GLOBALCONSTANTS myOpcUaAddresses (* Global constants *)
  (* Standard: 61499-1; Description: Copyright (c) 2026 Meisterschulen am Ostbahnhof This program and the accompanying materials are made available under the terms of the Eclipse Public License 2.0 which is available at https://www.eclipse.org/legal/epl-2.0/ SPDX-License-Identifier: EPL-2.0 *)
  (* Version 1.0, 2026-09-02, Franz Höpfinger, Meisterschulen am Ostbahnhof *)
  PACKAGE VV::const::OPC_UA;
  VAR_GLOBAL CONSTANT
    Q1_LOCAL_READ : WSTRING := "opc_ua[READ;/Objects/DigitalOutput/Q1,1:s=Output_Q1]"; (* Geraet B (Station 12): lokal ueberwachter Knoten fuer Output_Q1 (ACTION=READ, passend zu AX_SUBSCRIBE_1 - siehe 4diac-Doku opcua.adoc Tabelle: Local/READ/SUBSCRIBE), von Geraet A per CLIENT_1_0 remote beschrieben *)
    Q1_REMOTE_WRITE : WSTRING := "opc_ua[WRITE;opc.tcp://192.168.1.12:4840#;/Objects/DigitalOutput/Q1,1:s=Output_Q1]"; (* Geraet A (Station 11): aktiver Remote-Write ueber CLIENT_1_0 auf denselben Knoten wie Q1_LOCAL_READ auf Geraet B (ACTION=WRITE, passend zu CLIENT - Remote/WRITE/CLIENT) - Pfad/Name-Suffix muss identisch bleiben, IP muss als Literal dupliziert werden (kein Verweis auf Computers.gcf moeglich) *)
    FF1_TRIGGER_LOCAL_READ : WSTRING := "opc_ua[READ;/Objects/ToggleFF/FF1_Trigger,1:s=FF1_Trigger]"; (* Geraet B (Station 12): lokal ueberwachter Trigger-Knoten (ACTION=READ, passend zu AX_SUBSCRIBE_1 - Local/READ/SUBSCRIBE), von Geraet A per CLIENT_1_0 remote beschrieben, um SoftKey_F1-Tastendruecke ueber die Geraetegrenze zu takten *)
    FF1_TRIGGER_REMOTE_WRITE : WSTRING := "opc_ua[WRITE;opc.tcp://192.168.1.12:4840#;/Objects/ToggleFF/FF1_Trigger,1:s=FF1_Trigger]"; (* Geraet A (Station 11): aktiver Remote-Write ueber CLIENT_1_0 auf denselben Knoten wie FF1_TRIGGER_LOCAL_READ auf Geraet B (ACTION=WRITE, passend zu CLIENT - Remote/WRITE/CLIENT) - Pfad/Name-Suffix muss identisch bleiben, IP muss als Literal dupliziert werden *)
    FF1_STATE_LOCAL_READ : WSTRING := "opc_ua[READ;/Objects/ToggleFF/FF1_State,1:s=FF1_State]"; (* Geraet A (Station 11): lokal ueberwachter Flipflop-Zustandsknoten (ACTION=READ, passend zu AX_SUBSCRIBE_1 - Local/READ/SUBSCRIBE), von Geraet B per CLIENT_1_0 remote beschrieben, speist GreenWhiteBackground *)
    FF1_STATE_REMOTE_WRITE : WSTRING := "opc_ua[WRITE;opc.tcp://192.168.1.11:4840#;/Objects/ToggleFF/FF1_State,1:s=FF1_State]"; (* Geraet B (Station 12): aktiver Remote-Write ueber CLIENT_1_0 auf denselben Knoten wie FF1_STATE_LOCAL_READ auf Geraet A (ACTION=WRITE, passend zu CLIENT - Remote/WRITE/CLIENT) - Pfad/Name-Suffix muss identisch bleiben, IP muss als Literal dupliziert werden *)
  END_VAR
END_GLOBALCONSTANTS
